FUNCTION_BLOCK FB_StationBin
VAR_INPUT
	bEnableBin			: BOOL; // input for Enable Bin 
	Home_Sensor 		: BOOL; // input for home
	Safe_Sensor 		: BOOL;	// input for safe
	Dispense_Sensor 	: BOOL; // input for dispense
	Part_Present		: BOOL; // input for part present
	Dependency_OK		: BOOL; // input to check for dependency
	At_Station			: BOOL; // Input for bowl at station, used for reset condition too
END_VAR
VAR_OUTPUT
	Trigger_Of_Drive	: BOOL;	// Output for Enable of drive movement
	Direction_OF_Drive	: BOOL; // Output for Direction of drive - TRUE- Direction Positive, False - Direction Negative
	Lock_Dependency		: BOOL; // Output for Lock Dependency
	Count_OF_Parts		: INT;	// Counting of loaded parts
	bError				: BOOL; // Station is in Error
	sStatus				: STRING(255); // Message
END_VAR
VAR_IN_OUT
	ResetPartCount		: BOOL;		// Reset Counter of parts
	ResetBin			: BOOL;		// Reset Bin Logic
END_VAR
VAR
	TimerTimeout		: TON; // Use for timeout
	
	// Times
	tTimeoutMoving		: TIME := T#5000MS;
	tTimeoutDispence	: TIME := T#2000MS;
	
	iStep				: INT; // Step of the machine logic
END_VAR

IF NOT bEnableBin THEN
	iStep := 0;
	bError := FALSE;
	sStatus := 'Waiting for bin Enable';
	Count_OF_Parts := 0;
	Lock_Dependency := FALSE;
	Trigger_Of_Drive := FALSE;
ELSE
	IF ResetPartCount THEN
		ResetPartCount := FALSE;
		Count_OF_Parts := 0;
	END_IF
	IF ResetBin THEN
		ResetBin := FALSE;
		iStep := 0;
		Count_OF_Parts := 0;
		Lock_Dependency := FALSE;
		Trigger_Of_Drive := FALSE;
	END_IF
	CASE iStep OF
		0:  // Waiting part on Home
			IF bError THEN
				bError := FALSE;
			END_IF
			sStatus := 'Waiting for Part on Home';
			IF Home_Sensor 
			AND Part_Present 
			THEN
				iStep := 10;
			END_IF
			
		10: // Move to Safe
			Trigger_Of_Drive := TRUE;
			Direction_OF_Drive := TRUE;
			iStep := 11;
			
		11: // Wait Safe Done
			TimerTimeout(IN := TRUE, PT:= tTimeoutMoving);
			IF Safe_Sensor THEN
				Trigger_Of_Drive := FALSE;
				TimerTimeout(IN := FALSE);
				iStep := 20;
			ELSIF TimerTimeout.Q THEN
				sStatus := 'Timeout When Going to Safe';
				iStep := 1000; // Error
			END_IF
		
		20: // Check Dependency OK
			sStatus := 'Waiting Dependency OK';
			IF Dependency_OK 
			AND AT_Station 
			THEN
				sStatus := 'Going to Dispense';
				Lock_Dependency := TRUE;
				iStep := 30;
			END_IF
		
		30: // Move to Dispense
			Trigger_Of_Drive := TRUE;
			Direction_OF_Drive := TRUE;
			iStep := 31;
			
		31: // Wait Dispense
			TimerTimeout(IN := TRUE, PT:= tTimeoutMoving);
			IF Dispense_Sensor THEN
				Trigger_Of_Drive := FALSE;
				TimerTimeout(IN := FALSE);
				iStep := 40;
			ELSIF TimerTimeout.Q THEN
				sStatus := 'Timeout When Going to Dispense';
				iStep := 1000; // Error
			END_IF
		
		40: // Check Dispense Done
			TimerTimeout(IN := TRUE, PT:= tTimeoutDispence);
			IF NOT Part_Present THEN
				Count_OF_Parts := Count_OF_Parts + 1;
				TimerTimeout(IN := FALSE);
				iStep := 50;
			ELSIF TimerTimeout.Q THEN
				sStatus := 'Timeout When Not Part Present - Dispense Done';
				iStep := 1000; // Error
			END_IF
			
		50: // Start Move back to Safety
			Trigger_Of_Drive := TRUE;
			Direction_OF_Drive := FALSE;
			iStep := 51;
			
		51: // Wait Move back to Safety
			TimerTimeout(IN := TRUE, PT:= tTimeoutMoving);
			IF Safe_Sensor THEN
				Trigger_Of_Drive := FALSE;
				Lock_Dependency := FALSE;
				TimerTimeout(IN := FALSE);
				iStep := 60;
			ELSIF TimerTimeout.Q THEN
				sStatus := 'Timeout When Going back to Safe';
				iStep := 1000; // Error
			END_IF
		
		60: // Start Move Back To Home
			Trigger_Of_Drive := TRUE;
			Direction_OF_Drive := FALSE;
			iStep := 61;
		
		61: // Wait Move Back to Home
			TimerTimeout(IN := TRUE, PT:= tTimeoutMoving);
			IF Home_Sensor THEN
				Trigger_Of_Drive := FALSE;
				TimerTimeout(IN := FALSE);
				iStep := 0;
			ELSIF TimerTimeout.Q THEN
				sStatus := 'Timeout When Going back to Safe';
				iStep := 1000; // Error
			END_IF	
			
		1000:
			bError := TRUE;
			Trigger_Of_Drive := FALSE;
			TimerTimeout(IN := FALSE);
	END_CASE
END_IF

END_FUNCTION_BLOCK

(* stored: Version 1.1.0.1, ProductVersion 3.1.4024.9
   POU FB_StationBin: Id {44b87a21-45c0-4835-aecf-5faccdf116c6}, SpecialFunc None *)
